// SIMATIC S7-200 project (STEP 7-Micro/WIN), CPU 224 REL 02.01

SYMBOL_TABLE USER1
start            I0.0
stopp            I0.1
s1               I0.2
s2               I0.3
bt1              Q0.0
bt2              Q0.1
END_SYMBOL_TABLE

ORGANIZATION_BLOCK MAIN:OB1
TITLE=PROGRAM COMMENTS
BEGIN
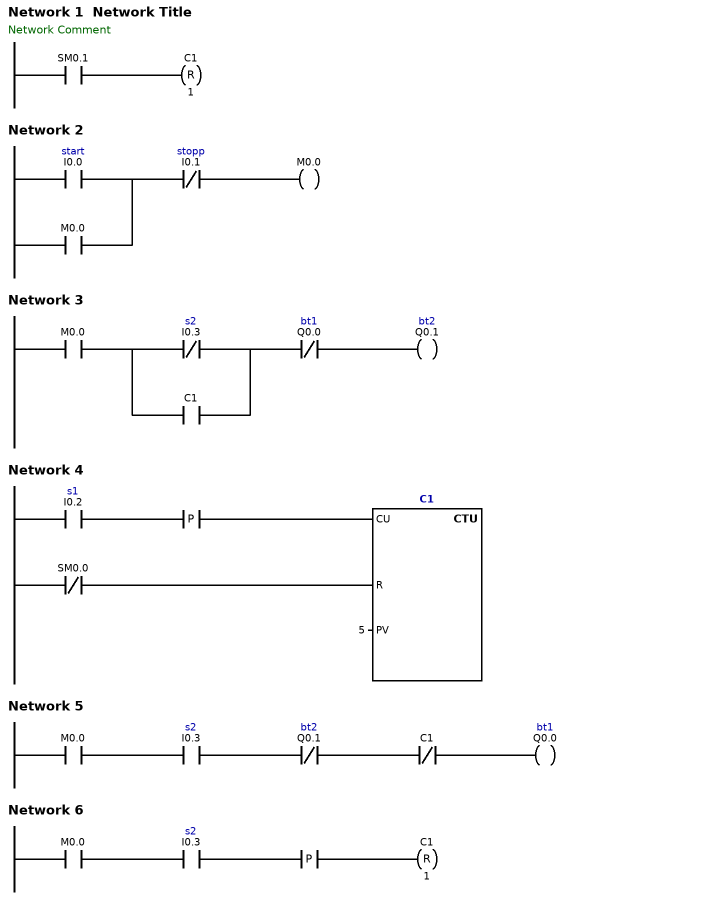
Network 1 // Network Title
// Network Comment
LD     SM0.1
R      C1, 1
Network 2
LD     start:I0.0
O      M0.0
AN     stopp:I0.1
=      M0.0
Network 3
LD     M0.0
LDN    s2:I0.3
O      C1
ALD
AN     bt1:Q0.0
=      bt2:Q0.1
Network 4
LD     s1:I0.2
EU
LDN    SM0.0
CTU    C1, 5
Network 5
LD     M0.0
A      s2:I0.3
AN     bt2:Q0.1
AN     C1
=      bt1:Q0.0
Network 6
LD     M0.0
A      s2:I0.3
EU
R      C1, 1
END_ORGANIZATION_BLOCK
